ABB RAPID module: Calibracion.mod

MODULE TCPZ_Tipjay
	! Points are read in order of declaration.
  ! Please do not change the order of points!

  LOCAL PERS robtarget pTCPZ_Point1:=[[-336.2762,-598.762,247.5795],[0.341533988714218,0.433732777833939,0.29114180803299,-0.781323730945587],[-2,-2,1,0],[9E+09,9E+09,9E+09,9E+09,9E+09,9E+09]];
	LOCAL PERS robtarget pTCPZ_Point2:=[[-331.8249,-603.8643,250.0889],[0.185168534517288,0.635887980461121,-0.232568770647049,-0.712229430675507],[-2,-2,1,0],[9E+09,9E+09,9E+09,9E+09,9E+09,9E+09]];
	LOCAL PERS robtarget pTCPZ_Point3:=[[-373.6251,-578.2554,239.8257],[0.398932665586472,0.70875096321106,-0.176154151558876,-0.554521799087524],[-2,-2,2,0],[9E+09,9E+09,9E+09,9E+09,9E+09,9E+09]];
	LOCAL PERS robtarget pTCPZ_Point4:=[[-336.9242,-584.8609,231.2205],[0.268533378839493,-0.21112123131752,0.80331015586853,-0.487863034009933],[-2,0,-3,0],[9E+09,9E+09,9E+09,9E+09,9E+09,9E+09]];
	LOCAL PERS robtarget pTCPZ_ElongZ:=[[-358.3258,-618.7408,270.9408],[0.313103079795837,0.597719788551331,0.33629247546196,-0.656966388225555],[-2,2,-3,0],[9E+09,9E+09,9E+09,9E+09,9E+09,9E+09]];
	TASK PERS tooldata Prueba:=[TRUE,[[82.1273,9.16203,35.9247],[0.353653,-0.00162473,0.935365,0.00429713]],[-1,[0,0,0],[1,0,0,0],0,0,0]];

ENDMODULE
